{attribute 'qualified_only'}
TYPE E_MMPathMotionStatus :
(
	eMMPathMotionStatus_Enabled				:= 0,																	(**)
	eMMPathMotionStatus_SuspendedByCommand	:= 1,																	(**)
	eMMPathMotionStatus_EStopActive			:= 2,																	(**)
	eMMPathMotionStatus_InterlockActive		:= 3																	(**)
) BYTE;
END_TYPE

(* stored: Version 1.1.0.1, ProductVersion 3.1.4024.5
   EnumerationTextList E_MMPathMotionStatus: Id {db46d0c4-62c5-4f6a-8cf2-afd32a662f37} *)
